// TIA Portal V15.1 export
// export: Created 2024-05-17T05:38:13.9331054Z, ExportSetting WithDefaults, DisplayName Totally Integrated Automation Portal, DisplayVersion V15.1 Update 5, DisplayName TIA Portal Openness, DisplayVersion V15.1 Update 5, DisplayName SINAMICS Startdrive Advanced, DisplayVersion V15.1, DisplayName G130, G150, S120, S150, SINAMICS MV, S210, DisplayVersion V15.1, DisplayName G110M, G120, G120C, G120D, G120P, DisplayVersion V15.1, DisplayName STEP 7 Professional, DisplayVersion V15.1 Update 5, DisplayName STEP 7 Safety, DisplayVersion V15.1, DisplayName WinCC Professional, DisplayVersion V15.1 Update 5, DisplayName SIMATIC Visualization Architect, DisplayVersion V15.1
DATA_BLOCK "_209210ZS01Passiv"   // DB323
{ S7_Optimized_Access := 'FALSE' }
AUTHOR : VCC
VERSION : 0.1
// stored: AutoNumber false, DBAccessibleFromOPCUA true, IsOnlyStoredInLoadMemory false, IsWriteProtectedInAS false
   VAR RETAIN
      AA_209000AK03JX36QF5240 { ExternalAccessible := 'False'; ExternalVisible := 'False'; ExternalWritable := 'False'} : Bool;   // Passivation alarm - ET200sp I/O - Safety Card QF5240
      AA_209000AK03JX36QF5246 { ExternalAccessible := 'False'; ExternalVisible := 'False'; ExternalWritable := 'False'} : Bool;   // Passivation alarm - ET200sp I/O - Safety Card QF5246
      AA_209210AS10JX40IF5400 { ExternalAccessible := 'False'; ExternalVisible := 'False'; ExternalWritable := 'False'} : Bool;   // Passivation alarm - ET200sp I/O - Safety Card IF5400
      AA_209210AX01JX41IF5450 { ExternalAccessible := 'False'; ExternalVisible := 'False'; ExternalWritable := 'False'} : Bool;   // Passivation alarm - ET200sp I/O - Safety Card IF5450
      AA_209210AS11JX42IF5500 { ExternalAccessible := 'False'; ExternalVisible := 'False'; ExternalWritable := 'False'} : Bool;   // Passivation alarm - ET200sp I/O - Safety Card IF5500
      AA_209210AX02JX43IF5550 { ExternalAccessible := 'False'; ExternalVisible := 'False'; ExternalWritable := 'False'} : Bool;   // Passivation alarm - ET200sp I/O - Safety Card IF5550
      AA_209210AS20JX48IF5600 { ExternalAccessible := 'False'; ExternalVisible := 'False'; ExternalWritable := 'False'} : Bool;   // Passivation alarm - ET200sp I/O - Safety Card IF5600
      AA_209000AK03M1UE130 { ExternalAccessible := 'False'; ExternalVisible := 'False'; ExternalWritable := 'False'} : Bool;   // Passivation alarm - MoviDrive - 210CR21M1
      AA_209000AK03M4UE131 { ExternalAccessible := 'False'; ExternalVisible := 'False'; ExternalWritable := 'False'} : Bool;   // Passivation alarm - MoviDrive - 210CS22M4ME1 (Power)
      AA_209000AK03M4UE132 { ExternalAccessible := 'False'; ExternalVisible := 'False'; ExternalWritable := 'False'} : Bool;   // Passivation alarm - MoviDrive - 210CS22M4ME2 (Brake)
      AA_209000AK03M1UE133 { ExternalAccessible := 'False'; ExternalVisible := 'False'; ExternalWritable := 'False'} : Bool;   // Passivation alarm - MoviDrive - 210CR23M1
      AA_209210CHB21M14UE134 { ExternalAccessible := 'False'; ExternalVisible := 'False'; ExternalWritable := 'False'} : Bool;   // Passivation alarm - MoviFit - 210CHB21M14
      "209000AK03JX36QF5240AlarmABCondition" { ExternalAccessible := 'False'; ExternalVisible := 'False'; ExternalWritable := 'False'} : Bool;   // Alarm AB condition
      "209000AK03JX36QF5246AlarmABCondition" { ExternalAccessible := 'False'; ExternalVisible := 'False'; ExternalWritable := 'False'} : Bool;   // Alarm AB condition
      "209210AS10JX40IF5400AlarmABCondition" { ExternalAccessible := 'False'; ExternalVisible := 'False'; ExternalWritable := 'False'} : Bool;   // Alarm AB condition
      "209210AX01JX41IF5450AlarmABCondition" { ExternalAccessible := 'False'; ExternalVisible := 'False'; ExternalWritable := 'False'} : Bool;   // Alarm AB condition
      "209210AS11JX42IF5500AlarmABCondition" { ExternalAccessible := 'False'; ExternalVisible := 'False'; ExternalWritable := 'False'} : Bool;   // Alarm AB condition
      "209210AX02JX43IF5550AlarmABCondition" { ExternalAccessible := 'False'; ExternalVisible := 'False'; ExternalWritable := 'False'} : Bool;   // Alarm AB condition
      "209210AS20JX48IF5600AlarmABCondition" { ExternalAccessible := 'False'; ExternalVisible := 'False'; ExternalWritable := 'False'} : Bool;   // Alarm AB condition
      "209000AK03M1UE130AlarmABCondition" { ExternalAccessible := 'False'; ExternalVisible := 'False'; ExternalWritable := 'False'} : Bool;   // Alarm AB condition
      "209000AK03M4UE131AlarmABCondition" { ExternalAccessible := 'False'; ExternalVisible := 'False'; ExternalWritable := 'False'} : Bool;   // Alarm AB condition
      "209000AK03M4UE132AlarmABCondition" { ExternalAccessible := 'False'; ExternalVisible := 'False'; ExternalWritable := 'False'} : Bool;   // Alarm AB condition
      "209000AK03M1UE133AlarmABCondition" { ExternalAccessible := 'False'; ExternalVisible := 'False'; ExternalWritable := 'False'} : Bool;   // Alarm AB condition
      "209210CHB21M14UE134AlarmABCondition" { ExternalAccessible := 'False'; ExternalVisible := 'False'; ExternalWritable := 'False'} : Bool;   // Alarm AB condition
      H_209000AK03JX36QF5240IAnim : Word;   // HMI Animation of the icon
      H_209000AK03JX36QF5246IAnim : Word;   // HMI Animation of the icon
      H_209210AS10JX40IF5400IAnim : Word;   // HMI Animation of the icon
      H_209210AX01JX41IF5450IAnim : Word;   // HMI Animation of the icon
      H_209210AS11JX42IF5500IAnim : Word;   // HMI Animation of the icon
      H_209210AX02JX43IF5550IAnim : Word;   // HMI Animation of the icon
      H_209210AS20JX48IF5600IAnim : Word;   // HMI Animation of the icon
      H_209000AK03M1UE130IAnim : Word;   // HMI Animation of the icon
      H_209000AK03M4UE131IAnim : Word;   // HMI Animation of the icon
      H_209000AK03M4UE132IAnim : Word;   // HMI Animation of the icon
      H_209000AK03M1UE133IAnim : Word;   // HMI Animation of the icon
      H_209210CHB21M14UE134IAnim : Word;   // HMI Animation of the icon
      H_Anim : Word;   // Animation
      H_DBnr : Int;   // DB number
      AlarmA { ExternalAccessible := 'False'; ExternalVisible := 'False'; ExternalWritable := 'False'} : Bool;   // Summary Alarm A
      AlarmB { ExternalAccessible := 'False'; ExternalVisible := 'False'; ExternalWritable := 'False'} : Bool;   // Summary Alarm B
      AlarmC { ExternalAccessible := 'False'; ExternalVisible := 'False'; ExternalWritable := 'False'} : Bool;   // Summary Alarm C
      AlarmD { ExternalAccessible := 'False'; ExternalVisible := 'False'; ExternalWritable := 'False'} : Bool;   // Summary Alarm D
      AlarmABCondition { ExternalAccessible := 'False'; ExternalVisible := 'False'; ExternalWritable := 'False'} : Bool;   // Alarm AB Condition
      PassivationError { ExternalAccessible := 'False'; ExternalVisible := 'False'; ExternalWritable := 'False'} : Bool;   // There is one ore more Passivation Errors active
      FeedBackError { ExternalAccessible := 'False'; ExternalVisible := 'False'; ExternalWritable := 'False'} : Bool;   // There is one ore more FeedBack Errors active
      "AckReqSendRcvDP/PN" { ExternalAccessible := 'False'; ExternalVisible := 'False'; ExternalWritable := 'False'} : Bool;   // Ack.Req from DP/DP or PN/PN couplers
   END_VAR
BEGIN
END_DATA_BLOCK
